  rq_activate_all_grippers(False)
  # end: URCap Program Node
  end
  thread Gripper_Activate_thread():
  Gripper_Activate_definition()
  daemon.done_executing()
  end
  def Gripper_Activate():
  textmsg("Executing event: Gripper_Activate")
  __er_thread_handle = run Gripper_Activate_thread()
  end
  if (not daemon.register_method("Gripper_Activate","[]", False)):
    textmsg("Failed to connect to register method Gripper_Activate")
    halt
  end
  sync()
  # end: URCap Program Node
  # begin: URCap Program Node
  #   Source: EnabledRobotics - ER-ABILITY, 5.0.0, Enabled Robotics ApS
  #   Type: EventNode
  $ 10 "EventNode: Gripper_Open1" "noBreak"
  def Gripper_Open1_definition():
  # begin: URCap Program Node
  #   Source: Robotiq_Grippers, 1.8.13.22852, Robotiq Inc.
  #   Type: Gripper
  $ 11 "Gripper Open (1)" "noBreak"
  if not(gripper_connected[0]):
    popup("Gripper 1 must be connected to run this program.", "No connection", False, True, True)
  end
  if not(rq_is_gripper_activated("1")):
    popup("Gripper 1 is not activated. Go to Installation tab > Gripper to activate it and run the program again.", "Not activated", False, True, True)
  end
  rq_set_pos_spd_for(0, 255, 0, "1")
  rq_wait_pos_spe_for_request(0, 255, 0, "1")
  rq_go_to("1")
  rq_wait("1")
  # end: URCap Program Node
  end
  thread Gripper_Open1_thread():
  Gripper_Open1_definition()
  daemon.done_executing()
  end
  def Gripper_Open1():
  textmsg("Executing event: Gripper_Open1")
  __er_thread_handle = run Gripper_Open1_thread()
  end
  if (not daemon.register_method("Gripper_Open1","[]", False)):
    textmsg("Failed to connect to register method Gripper_Open1")
    halt
  end
  sync()
  # end: URCap Program Node
  # begin: URCap Program Node
  #   Source: EnabledRobotics - ER-ABILITY, 5.0.0, Enabled Robotics ApS
  #   Type: EventNode
  $ 12 "EventNode: Gripper_Close" "noBreak"
  def Gripper_Close_definition():
  # begin: URCap Program Node
  #   Source: Robotiq_Grippers, 1.8.13.22852, Robotiq Inc.
  #   Type: Gripper
  $ 13 "Gripper Close (1)" "noBreak"
  if not(gripper_connected[0]):
    popup("Gripper 1 must be connected to run this program.", "No connection", False, True, True)
  end
  if not(rq_is_gripper_activated("1")):
    popup("Gripper 1 is not activated. Go to Installation tab > Gripper to activate it and run the program again.", "Not activated", False, True, True)
  end
  rq_set_pos_spd_for(255, 255, 0, "1")
  rq_wait_pos_spe_for_request(255, 255, 0, "1")
  rq_go_to("1")
  rq_wait("1")
  # end: URCap Program Node
  end
  thread Gripper_Close_thread():
  Gripper_Close_definition()
  daemon.done_executing()
  end
  def Gripper_Close():
  textmsg("Executing event: Gripper_Close")
  __er_thread_handle = run Gripper_Close_thread()
  end
  if (not daemon.register_method("Gripper_Close","[]", False)):
    textmsg("Failed to connect to register method Gripper_Close")
    halt
  end
  sync()
  # end: URCap Program Node
  # begin: URCap Program Node
  #   Source: EnabledRobotics - ER-ABILITY, 5.0.0, Enabled Robotics ApS
  #   Type: EventNode
  $ 14 "EventNode: Unload" "noBreak"
  global __er_Unload_arg_pose = p[0, 0, 0, 0, 0, 0]
  def Unload_definition(arg_pose):
  $ 15 "Unload_ref≔__er_Unload_arg_pose" "noBreak"
  global Unload_ref=__er_Unload_arg_pose
  $ 16 "MoveJ" "noBreak"
  $ 17 "Waypoint_2" "noBreak"
  movej(get_inverse_kin(Waypoint_2_p, qnear=Waypoint_2_q), a=1.3962634015954636, v=1.0471975511965976)
  $ 18 "Pallet_2" "noBreak"
  def Pallet_2_trans(pose):
  return p[pose[0], pose[1], pose[2], 0, 0, 0]
  end
  def Pallet_2_rot(pose):
  return p[0, 0, 0, pose[3], pose[4], pose[5]]
  end
  def Pallet_2_compute_pallet_waypoint(T_base_feature_taught, T_feature_referencePoint_taught, T_referencePoint_approach_taught, T_base_feature, T_base_referencePoint):
  local trans_referencePoint_approach_in_feature_taught = pose_sub(Pallet_2_trans(pose_trans(T_feature_referencePoint_taught, T_referencePoint_approach_taught)), Pallet_2_trans(T_feature_referencePoint_taught))
  local rot_referencePoint_approach_in_feature_taught = pose_trans(Pallet_2_rot(T_feature_referencePoint_taught), pose_trans(Pallet_2_rot(T_referencePoint_approach_taught), pose_inv(Pallet_2_rot(T_feature_referencePoint_taught))))
  T_feature_referencePoint = pose_trans(pose_inv(T_base_feature), T_base_referencePoint)
  rot_referencePoint_approach = pose_trans(pose_inv(Pallet_2_rot(T_feature_referencePoint)), pose_trans(rot_referencePoint_approach_in_feature_taught, Pallet_2_rot(T_feature_referencePoint)))
  T_feature_approach = pose_trans(trans_referencePoint_approach_in_feature_taught, pose_trans(T_feature_referencePoint, rot_referencePoint_approach))
  T_base_approach = pose_trans(T_base_feature, T_feature_approach)
  return T_base_approach
  end
  Pallet_2_tct_1 = 3
  if (Pallet_2_cnt_1 > 3 or Pallet_2_cnt_1 < 1):
    Pallet_2_cnt_1 = 1
  end
  $ 19 "Patterns" "noBreak"
  $ 20 "Line_Pattern_2" "noBreak"
  $ 23 "Layers" "noBreak"
  if (Pallet_2_cnt_1 < 4):
    Pallet_2_lno_1 = 1
    Pallet_2_lct_1 = Pallet_2_cnt_1
    global StartItem_2=pose_trans(p[0.0,0.0,0.0,0.0,0.0,0.0], pose_trans(p[-.000000000000, -.000000000000, -.000000000000, .000000000000, .000000000000, .000000000000], p[.520226808930, .071936160165, -.439816599331, 3.141509651494, .015551157232, .000010800258]))
    global EndItem_2=pose_trans(p[0.0,0.0,0.0,0.0,0.0,0.0], pose_trans(p[-.000000000000, -.000000000000, -.000000000000, .000000000000, .000000000000, .000000000000], p[.521976506042, -.107892547401, -.439624527362, 3.141328655500, .039596804554, -.000022510547]))
    referencePoint = interpolate_pose(StartItem_2, EndItem_2, (Pallet_2_lct_1 - 1)/2)
    if ((Pallet_2_lct_1 - 1) < 1.5):
      qNearApproach = [2.5448785455331526, 0.32353681292985914, 0.8867449467631632, -1.209835749483231, -0.6015755965885301, -3.1422033514088064]
    else:
      qNearApproach = [2.318553773487707, 0.5230815444746025, 0.3070377710571135, -0.8290774467610227, -0.8454805618969878, -3.143220671816902]
    end
    direction = p[0,0,1,0,0,0]
    referencePoint = pose_add (referencePoint,p[0.0*direction[0],0.0*direction[1],0.0*direction[2],0,0,0])
  end
  Approach_3_p = Pallet_2_compute_pallet_waypoint(p[0.0,0.0,0.0,0.0,0.0,0.0], pose_trans(pose_inv(p[0.0,0.0,0.0,0.0,0.0,0.0]), p[0.52022680893046,0.07193616016490022,-0.4398165993312858,3.1415096514942586,0.01555115723185833,1.080025776929912E-5]), p[-1.5009913569219435E-4,-1.4773289497117814E-4,-0.07363840846726544,4.5745872302844587E-4,-5.141193914981974E-4,-2.8251868715170223E-4], p[0.0,0.0,0.0,0.0,0.0,0.0], referencePoint)
  Approach_3_p = pose_trans(p[0.52022680893046,0.07193616016490022,-0.4398165993312858,3.141509651511718,0.015551157231944729,1.0800257734370728E-5], pose_trans(pose_inv(referencePoint), Approach_3_p))
  Approach_3_q = qNearApproach
  ToolActionPoi_3_p = Pallet_2_compute_pallet_waypoint(p[0.0,0.0,0.0,0.0,0.0,0.0], pose_trans(pose_inv(p[0.0,0.0,0.0,0.0,0.0,0.0]), p[0.52022680893046,0.07193616016490022,-0.4398165993312858,3.1415096514942586,0.01555115723185833,1.080025776929912E-5]), p[-1.1102230246251565E-16,1.3877787807814457E-17,0.0,0.0,0.0,0.0], p[0.0,0.0,0.0,0.0,0.0,0.0], referencePoint)
  ToolActionPoi_3_p = pose_trans(p[0.52022680893046,0.07193616016490022,-0.4398165993312858,3.141509651511718,0.015551157231944729,1.0800257734370728E-5], pose_trans(pose_inv(referencePoint), ToolActionPoi_3_p))
  Exit_4_p = Pallet_2_compute_pallet_waypoint(p[0.0,0.0,0.0,0.0,0.0,0.0], pose_trans(pose_inv(p[0.0,0.0,0.0,0.0,0.0,0.0]), p[0.52022680893046,0.07193616016490022,-0.4398165993312858,3.1415096514942586,0.01555115723185833,1.080025776929912E-5]), p[-3.93932843645306E-6,-7.071115271761741E-6,-0.10081098319262166,2.4279295122529868E-5,-8.605183831750915E-6,-1.5904010148868937E-5], p[0.0,0.0,0.0,0.0,0.0,0.0], referencePoint)
  Exit_4_p = pose_trans(p[0.52022680893046,0.07193616016490022,-0.4398165993312858,3.141509651511718,0.015551157231944729,1.0800257734370728E-5], pose_trans(pose_inv(referencePoint), Exit_4_p))
  $ 24 "At Each Item" "noBreak"
  $ 25 "Generated Movements" "noBreak"
  $ 26 "MoveJ" "noBreak"
  $ 27 "Approach_3" "noBreak"
  movej(get_inverse_kin(pose_trans(referencePoint, pose_trans(p[-.520910568349, .066801880452, -.439817090922, -3.141509651507, -.015551157232, -.000010800258], Approach_3_p)), qnear=Approach_3_q), a=1.3962634015954636, v=1.0471975511965976)
  $ 28 "MoveL" "noBreak"
  $ 29 "ToolActionPoi_3" "noBreak"
  movel(pose_trans(referencePoint, pose_trans(p[-.520910568349, .066801880452, -.439817090922, -3.141509651507, -.015551157232, -.000010800258], ToolActionPoi_3_p)), a=1.2, v=0.25)
  $ 30 "Tool action" "noBreak"
  # begin: URCap Program Node
  #   Source: Robotiq_Grippers, 1.8.13.22852, Robotiq Inc.
  #   Type: Gripper
  $ 31 "Gripper Close (1)" "noBreak"
  if not(gripper_connected[0]):
    popup("Gripper 1 must be connected to run this program.", "No connection", False, True, True)
  end
  if not(rq_is_gripper_activated("1")):
    popup("Gripper 1 is not activated. Go to Installation tab > Gripper to activate it and run the program again.", "Not activated", False, True, True)
  end
  rq_set_pos_spd_for(255, 255, 255, "1")
  rq_wait_pos_spe_for_request(255, 255, 255, "1")
  rq_go_to("1")
  rq_wait("1")
  # end: URCap Program Node
  $ 32 "MoveL" "noBreak"
  $ 33 "Exit_4" "noBreak"
  movel(pose_trans(referencePoint, pose_trans(p[-.520910568349, .066801880452, -.439817090922, -3.141509651507, -.015551157232, -.000010800258], Exit_4_p)), a=1.2, v=0.25)
  Pallet_2_sep_1 = False
  if (Pallet_2_cnt_1 >= 3):
    Pallet_2_cnt_1 = 1
  else:
    Pallet_2_cnt_1 = Pallet_2_cnt_1 + 1
  end
  $ 34 "MoveJ" "noBreak"
  $ 35 "Waypoint_2" "noBreak"
  movej(get_inverse_kin(Waypoint_2_p, qnear=Waypoint_2_q), a=1.3962634015954636, v=1.0471975511965976)
  $ 36 "Pallet_1" "noBreak"
  def Pallet_1_trans(pose):
  return p[pose[0], pose[1], pose[2], 0, 0, 0]
  end
  def Pallet_1_rot(pose):
  return p[0, 0, 0, pose[3], pose[4], pose[5]]
  end
  def Pallet_1_compute_pallet_waypoint(T_base_feature_taught, T_feature_referencePoint_taught, T_referencePoint_approach_taught, T_base_feature, T_base_referencePoint):
  local trans_referencePoint_approach_in_feature_taught = pose_sub(Pallet_1_trans(pose_trans(T_feature_referencePoint_taught, T_referencePoint_approach_taught)), Pallet_1_trans(T_feature_referencePoint_taught))
  local rot_referencePoint_approach_in_feature_taught = pose_trans(Pallet_1_rot(T_feature_referencePoint_taught), pose_trans(Pallet_1_rot(T_referencePoint_approach_taught), pose_inv(Pallet_1_rot(T_feature_referencePoint_taught))))
  T_feature_referencePoint = pose_trans(pose_inv(T_base_feature), T_base_referencePoint)
  rot_referencePoint_approach = pose_trans(pose_inv(Pallet_1_rot(T_feature_referencePoint)), pose_trans(rot_referencePoint_approach_in_feature_taught, Pallet_1_rot(T_feature_referencePoint)))
  T_feature_approach = pose_trans(trans_referencePoint_approach_in_feature_taught, pose_trans(T_feature_referencePoint, rot_referencePoint_approach))
  T_base_approach = pose_trans(T_base_feature, T_feature_approach)
  return T_base_approach
  end
  Pallet_2_tct_2 = 3
  if (Pallet_2_cnt_2 > 3 or Pallet_2_cnt_2 < 1):
    Pallet_2_cnt_2 = 1
  end
  $ 37 "Patterns" "noBreak"
  $ 38 "Line_Pattern_1" "noBreak"
  $ 41 "Layers" "noBreak"
  if (Pallet_2_cnt_2 < 4):
    Pallet_2_lno_2 = 1
    Pallet_2_lct_2 = Pallet_2_cnt_2
    global StartItem_1=pose_trans(Unload_ref, pose_trans(p[-.592420775083, .276699022305, .196891037220, 2.141026582984, -2.289780745210, -.016012414057], p[.145742456500, -.623712299717, .141843363677, -2.162912830523, 2.278464349970, .000016883489]))
    global EndItem_1=pose_trans(Unload_ref, pose_trans(p[-.592420775083, .276699022305, .196891037220, 2.141026582984, -2.289780745210, -.016012414057], p[-.034366509976, -.616405446345, .140307709095, 2.162884038701, -2.278479638159, .000010711089]))
    referencePoin_1 = interpolate_pose(StartItem_1, EndItem_1, (Pallet_2_lct_2 - 1)/2)
    if ((Pallet_2_lct_2 - 1) < 1.5):
      qNearApproach_1 = [1.4717269593278084, -0.377092883754063, 1.1086358557351508, -4.010618644468483, 0.2053468506389249, 0.11347314803018159]
    else:
      qNearApproach_1 = [1.223852267476565, -0.3417190093073499, 1.0145159265446688, -3.879360012423625, 0.4524234852589557, 0.035990198425167035]
    end
    direction = pose_trans(p[0,0,0,Unload_ref[3],Unload_ref[4],Unload_ref[5]], p[0,0,1,0,0,0])
    referencePoin_1 = pose_add (referencePoin_1,p[0.0*direction[0],0.0*direction[1],0.0*direction[2],0,0,0])
  end
  Approach_p = Pallet_1_compute_pallet_waypoint(p[0.23673981765789284,-0.611972183808765,0.18903732227235456,-2.141026582984071,2.2897807452097325,0.016012414057338102], pose_trans(pose_inv(p[0.23673981765789284,-0.611972183808765,0.18903732227235456,-2.141026582984071,2.2897807452097325,0.016012414057338102]), p[0.14574245649996154,-0.6237122997166273,0.14184336367685696,-2.1629128305231067,2.278464349969941,1.688348907601959E-5]), p[0.0011206971510525632,0.0015926661309434986,-0.05760783126324068,0.031976489334781005,-0.019679141912164282,-0.020960074111678773], Unload_ref, referencePoin_1)
  Approach_p = pose_trans(p[0.3302161821107999,-0.6547625956979264,0.14667608988337466,2.3106327262625443,-2.073456813515827,-0.009785998864891442], pose_trans(pose_inv(referencePoin_1), Approach_p))
  Approach_q = qNearApproach_1
  ToolActionPoint_p = Pallet_1_compute_pallet_waypoint(p[0.23673981765789284,-0.611972183808765,0.18903732227235456,-2.141026582984071,2.2897807452097325,0.016012414057338102], pose_trans(pose_inv(p[0.23673981765789284,-0.611972183808765,0.18903732227235456,-2.141026582984071,2.2897807452097325,0.016012414057338102]), p[0.14574245649996154,-0.6237122997166273,0.14184336367685696,-2.1629128305231067,2.278464349969941,1.688348907601959E-5]), p[-0.05091451474589437,0.1798191171068455,0.009530418404298385,0.030088811758342437,-0.022546045786153587,0.16009642489347953], Unload_ref, referencePoin_1)
  ToolActionPoint_p = pose_trans(p[0.3302161821107999,-0.6547625956979264,0.14667608988337466,2.3106327262625443,-2.073456813515827,-0.009785998864891442], pose_trans(pose_inv(referencePoin_1), ToolActionPoint_p))
  Exit_1_p = Pallet_1_compute_pallet_waypoint(p[0.23673981765789284,-0.611972183808765,0.18903732227235456,-2.141026582984071,2.2897807452097325,0.016012414057338102], pose_trans(pose_inv(p[0.23673981765789284,-0.611972183808765,0.18903732227235456,-2.141026582984071,2.2897807452097325,0.016012414057338102]), p[0.14574245649996154,-0.6237122997166273,0.14184336367685696,-2.1629128305231067,2.278464349969941,1.688348907601959E-5]), p[0.0012088044817964994,6.156659549959032E-4,-0.05405850596043982,1.6947789472419606E-5,2.6304475016522655E-5,-6.152303689366298E-6], Unload_ref, referencePoin_1)
  Exit_1_p = pose_trans(p[0.3302161821107999,-0.6547625956979264,0.14667608988337466,2.3106327262625443,-2.073456813515827,-0.009785998864891442], pose_trans(pose_inv(referencePoin_1), Exit_1_p))
  $ 42 "At Each Item" "noBreak"
  $ 43 "Generated Movements" "noBreak"
  $ 44 "MoveJ" "noBreak"
  $ 45 "Approach" "noBreak"
  movej(get_inverse_kin(pose_trans(referencePoin_1, pose_trans(p[-.689448135507, .253081536651, .141002351928, -2.310632726263, 2.073456813516, .009785998865], Approach_p)), qnear=Approach_q), a=1.3962634015954636, v=1.0471975511965976)
  $ 46 "MoveL" "noBreak"
  $ 47 "ToolActionPoint" "noBreak"
  movel(pose_trans(referencePoin_1, pose_trans(p[-.689448135507, .253081536651, .141002351928, -2.310632726263, 2.073456813516, .009785998865], ToolActionPoint_p)), a=1.2, v=0.25)
  $ 48 "Tool action" "noBreak"
  # begin: URCap Program Node
  #   Source: Robotiq_Grippers, 1.8.13.22852, Robotiq Inc.
  #   Type: Gripper
  $ 49 "Gripper Open (1)" "noBreak"
  if not(gripper_connected[0]):
    popup("Gripper 1 must be connected to run this program.", "No connection", False, True, True)
  end
  if not(rq_is_gripper_activated("1")):
    popup("Gripper 1 is not activated. Go to Installation tab > Gripper to activate it and run the program again.", "Not activated", False, True, True)
  end
  rq_set_pos_spd_for(0, 255, 255, "1")
  rq_wait_pos_spe_for_request(0, 255, 255, "1")
  rq_go_to("1")
  rq_wait("1")
  # end: URCap Program Node
  $ 50 "MoveL" "noBreak"
  $ 51 "Exit_1" "noBreak"
  movel(pose_trans(referencePoin_1, pose_trans(p[-.689448135507, .253081536651, .141002351928, -2.310632726263, 2.073456813516, .009785998865], Exit_1_p)), a=1.2, v=0.25)
  Pallet_2_sep_2 = False
  if (Pallet_2_cnt_2 >= 3):
    Pallet_2_cnt_2 = 1
  else:
    Pallet_2_cnt_2 = Pallet_2_cnt_2 + 1
  end
  $ 52 "MoveJ" "noBreak"
  $ 53 "Waypoint_2" "noBreak"
  movej(get_inverse_kin(Waypoint_2_p, qnear=Waypoint_2_q), a=1.3962634015954636, v=1.0471975511965976)
  end
  thread Unload_thread():
  Unload_definition(__er_Unload_arg_pose)
  daemon.done_executing()
  end
  def Unload(arg_pose):
  textmsg("Executing event: Unload, with arguments:")
  textmsg("Argument: arg_pose = ", arg_pose)
  __er_Unload_arg_pose = arg_pose
  __er_thread_handle = run Unload_thread()
  end
  if (not daemon.register_method("Unload","[pose]", False)):
    textmsg("Failed to connect to register method Unload")
    halt
  end
  sync()
  # end: URCap Program Node
  # begin: URCap Program Node
  #   Source: EnabledRobotics - ER-ABILITY, 5.0.0, Enabled Robotics ApS
  #   Type: EventNode
  $ 54 "EventNode: Palletize" "noBreak"
  global __er_Palletize_arg_pose = p[0, 0, 0, 0, 0, 0]
  def Palletize_definition(arg_pose):
  $ 55 "Pallet_ref≔__er_Palletize_arg_pose" "noBreak"
  global Pallet_ref=__er_Palletize_arg_pose
  $ 56 "MoveJ" "noBreak"
  $ 58 "Waypoint_2" "noBreak"
  movej(get_inverse_kin(Waypoint_2_p, qnear=Waypoint_2_q), a=1.3962634015954636, v=1.0471975511965976)
  $ 59 "Pallet_3" "noBreak"
  def Pallet_3_trans(pose):
  return p[pose[0], pose[1], pose[2], 0, 0, 0]
  end
  def Pallet_3_rot(pose):
  return p[0, 0, 0, pose[3], pose[4], pose[5]]
  end
  def Pallet_3_compute_pallet_waypoint(T_base_feature_taught, T_feature_referencePoint_taught, T_referencePoint_approach_taught, T_base_feature, T_base_referencePoint):
  local trans_referencePoint_approach_in_feature_taught = pose_sub(Pallet_3_trans(pose_trans(T_feature_referencePoint_taught, T_referencePoint_approach_taught)), Pallet_3_trans(T_feature_referencePoint_taught))
  local rot_referencePoint_approach_in_feature_taught = pose_trans(Pallet_3_rot(T_feature_referencePoint_taught), pose_trans(Pallet_3_rot(T_referencePoint_approach_taught), pose_inv(Pallet_3_rot(T_feature_referencePoint_taught))))
  T_feature_referencePoint = pose_trans(pose_inv(T_base_feature), T_base_referencePoint)
  rot_referencePoint_approach = pose_trans(pose_inv(Pallet_3_rot(T_feature_referencePoint)), pose_trans(rot_referencePoint_approach_in_feature_taught, Pallet_3_rot(T_feature_referencePoint)))
  T_feature_approach = pose_trans(trans_referencePoint_approach_in_feature_taught, pose_trans(T_feature_referencePoint, rot_referencePoint_approach))
  T_base_approach = pose_trans(T_base_feature, T_feature_approach)
  return T_base_approach
  end
  Pallet_2_tct_3 = 3
  if (Pallet_2_cnt_3 > 3 or Pallet_2_cnt_3 < 1):
    Pallet_2_cnt_3 = 1
  end
  $ 60 "Patterns" "noBreak"
  $ 61 "Line_Pattern_5" "noBreak"
  $ 64 "Layers" "noBreak"
  if (Pallet_2_cnt_3 < 4):
    Pallet_2_lno_3 = 1
    Pallet_2_lct_3 = Pallet_2_cnt_3
    global StartItem_5=pose_trans(Pallet_ref, pose_trans(p[-.592420775083, .276699022305, .196891037220, 2.141026582984, -2.289780745210, -.016012414057], p[.145742456500, -.623712299717, .141843363677, -2.162912830523, 2.278464349970, .000016883489]))
    global EndItem_5=pose_trans(Pallet_ref, pose_trans(p[-.592420775083, .276699022305, .196891037220, 2.141026582984, -2.289780745210, -.016012414057], p[-.034364587449, -.616414812009, .134803893258, 2.162884771053, -2.278474941594, .000025529303]))
    referencePoin_6 = interpolate_pose(StartItem_5, EndItem_5, (Pallet_2_lct_3 - 1)/2)
    if ((Pallet_2_lct_3 - 1) < 1.5):
      qNearApproach_2 = [1.160836153948624, -0.48475985649287523, 1.429198472833832, -4.07612878433148, 0.3533404294143797, -0.011125824810111595]
    else:
      qNearApproach_2 = [0.9092989459402957, -0.3906363918532989, 1.217352351317741, -3.9632834025255583, 0.6055194004184299, -0.00720924811746837]
    end
    direction = pose_trans(p[0,0,0,Pallet_ref[3],Pallet_ref[4],Pallet_ref[5]], p[0,0,1,0,0,0])
    referencePoin_6 = pose_add (referencePoin_6,p[0.0*direction[0],0.0*direction[1],0.0*direction[2],0,0,0])
  end
  Approach_2_p = Pallet_3_compute_pallet_waypoint(p[0.23673981765789284,-0.611972183808765,0.18903732227235456,-2.141026582984071,2.2897807452097325,0.016012414057338102], pose_trans(pose_inv(p[0.23673981765789284,-0.611972183808765,0.18903732227235456,-2.141026582984071,2.2897807452097325,0.016012414057338102]), p[0.14574245649996154,-0.6237122997166273,0.14184336367685696,-2.1629128305231067,2.278464349969941,1.688348907601959E-5]), p[-8.821036119655012E-6,9.83391916484222E-6,-0.05174217287322935,-7.92077343834213E-7,-8.53904463359664E-6,4.718218270382111E-6], Pallet_ref, referencePoin_6)
  Approach_2_p = pose_trans(p[0.14574245649996245,-0.6237122997166271,0.14184336367685513,-2.162912830525248,2.2784643499679076,1.6883689364664383E-5], pose_trans(pose_inv(referencePoin_6), Approach_2_p))
  Approach_2_q = qNearApproach_2
  ToolActionPoi_2_p = Pallet_3_compute_pallet_waypoint(p[0.23673981765789284,-0.611972183808765,0.18903732227235456,-2.141026582984071,2.2897807452097325,0.016012414057338102], pose_trans(pose_inv(p[0.23673981765789284,-0.611972183808765,0.18903732227235456,-2.141026582984071,2.2897807452097325,0.016012414057338102]), p[0.14574245649996154,-0.6237122997166273,0.14184336367685696,-2.1629128305231067,2.278464349969941,1.688348907601959E-5]), p[2.220446049250313E-16,9.159339953157541E-16,-1.8318679906315083E-15,0.0,0.0,0.0], Pallet_ref, referencePoin_6)
  ToolActionPoi_2_p = pose_trans(p[0.14574245649996245,-0.6237122997166271,0.14184336367685513,-2.162912830525248,2.2784643499679076,1.6883689364664383E-5], pose_trans(pose_inv(referencePoin_6), ToolActionPoi_2_p))
  Exit_3_p = Pallet_3_compute_pallet_waypoint(p[0.23673981765789284,-0.611972183808765,0.18903732227235456,-2.141026582984071,2.2897807452097325,0.016012414057338102], pose_trans(pose_inv(p[0.23673981765789284,-0.611972183808765,0.18903732227235456,-2.141026582984071,2.2897807452097325,0.016012414057338102]), p[0.14574245649996154,-0.6237122997166273,0.14184336367685696,-2.1629128305231067,2.278464349969941,1.688348907601959E-5]), p[-4.6349033265835615E-6,6.324703609672522E-6,-0.06181962181018885,-2.875197051692597E-6,-4.847655252132371E-5,1.897897991802547E-5], Pallet_ref, referencePoin_6)
  Exit_3_p = pose_trans(p[0.33020295134031996,-0.6550358453350454,0.14679715883248884,2.3097137152461533,-2.071977896073306,-0.009558990049756003], pose_trans(pose_inv(referencePoin_6), Exit_3_p))
  $ 65 "At Each Item" "noBreak"
  $ 66 "Generated Movements" "noBreak"
  $ 67 "MoveJ" "noBreak"
  $ 68 "Approach_2" "noBreak"
  movej(get_inverse_kin(pose_trans(referencePoin_6, pose_trans(p[-.615288801215, .177976730796, .141849958260, 2.162912830677, -2.278464350127, -.000016883689], Approach_2_p)), qnear=Approach_2_q), a=1.3962634015954636, v=1.0471975511965976)
  $ 69 "MoveL" "noBreak"
  $ 70 "ToolActionPoi_2" "noBreak"
  movel(pose_trans(referencePoin_6, pose_trans(p[-.615288801215, .177976730796, .141849958260, 2.162912830677, -2.278464350127, -.000016883689], ToolActionPoi_2_p)), a=1.2, v=0.25)
  $ 71 "Tool action" "noBreak"
  # begin: URCap Program Node
  #   Source: Robotiq_Grippers, 1.8.13.22852, Robotiq Inc.
  #   Type: Gripper
  $ 72 "Gripper Close (1)" "noBreak"
  if not(gripper_connected[0]):
    popup("Gripper 1 must be connected to run this program.", "No connection", False, True, True)
  end
  if not(rq_is_gripper_activated("1")):
    popup("Gripper 1 is not activated. Go to Installation tab > Gripper to activate it and run the program again.", "Not activated", False, True, True)
  end
  rq_set_pos_spd_for(255, 153, 56, "1")
  rq_wait_pos_spe_for_request(255, 153, 56, "1")
  rq_go_to("1")
  rq_wait("1")
  # end: URCap Program Node
  $ 73 "MoveL" "noBreak"
  $ 74 "Exit_3" "noBreak"
  movel(pose_trans(referencePoin_6, pose_trans(p[-.689971033309, .252662774639, .140559059103, -2.309713715246, 2.071977896073, .009558990050], Exit_3_p)), a=1.2, v=0.25)
  Pallet_2_sep_3 = False
  if (Pallet_2_cnt_3 >= 3):
    Pallet_2_cnt_3 = 1
  else:
    Pallet_2_cnt_3 = Pallet_2_cnt_3 + 1
  end
  $ 75 "MoveJ" "noBreak"
  $ 76 "Waypoint_2" "noBreak"
  movej(get_inverse_kin(Waypoint_2_p, qnear=Waypoint_2_q), a=1.3962634015954636, v=1.0471975511965976)
  $ 77 "Pallet_4" "noBreak"
  def Pallet_4_trans(pose):
  return p[pose[0], pose[1], pose[2], 0, 0, 0]
  end
  def Pallet_4_rot(pose):
  return p[0, 0, 0, pose[3], pose[4], pose[5]]
  end
  def Pallet_4_compute_pallet_waypoint(T_base_feature_taught, T_feature_referencePoint_taught, T_referencePoint_approach_taught, T_base_feature, T_base_referencePoint):
  local trans_referencePoint_approach_in_feature_taught = pose_sub(Pallet_4_trans(pose_trans(T_feature_referencePoint_taught, T_referencePoint_approach_taught)), Pallet_4_trans(T_feature_referencePoint_taught))
  local rot_referencePoint_approach_in_feature_taught = pose_trans(Pallet_4_rot(T_feature_referencePoint_taught), pose_trans(Pallet_4_rot(T_referencePoint_approach_taught), pose_inv(Pallet_4_rot(T_feature_referencePoint_taught))))
  T_feature_referencePoint = pose_trans(pose_inv(T_base_feature), T_base_referencePoint)
  rot_referencePoint_approach = pose_trans(pose_inv(Pallet_4_rot(T_feature_referencePoint)), pose_trans(rot_referencePoint_approach_in_feature_taught, Pallet_4_rot(T_feature_referencePoint)))
  T_feature_approach = pose_trans(trans_referencePoint_approach_in_feature_taught, pose_trans(T_feature_referencePoint, rot_referencePoint_approach))
  T_base_approach = pose_trans(T_base_feature, T_feature_approach)
  return T_base_approach
  end
  Pallet_2_tct_4 = 3
  if (Pallet_2_cnt_4 > 3 or Pallet_2_cnt_4 < 1):
    Pallet_2_cnt_4 = 1
  end
  $ 78 "Patterns" "noBreak"
  $ 79 "Line_Pattern_6" "noBreak"
  $ 82 "Layers" "noBreak"
  if (Pallet_2_cnt_4 < 4):
    Pallet_2_lno_4 = 1
    Pallet_2_lct_4 = Pallet_2_cnt_4
    global StartItem_6=pose_trans(p[0.0,0.0,0.0,0.0,0.0,0.0], pose_trans(p[-.000000000000, -.000000000000, -.000000000000, .000000000000, .000000000000, .000000000000], p[.520226808930, .071936160165, -.439816599331, 3.141509651494, .015551157232, .000010800258]))
    global EndItem_6=pose_trans(p[0.0,0.0,0.0,0.0,0.0,0.0], pose_trans(p[-.000000000000, -.000000000000, -.000000000000, .000000000000, .000000000000, .000000000000], p[.521976506042, -.107892547401, -.439624527362, 3.141328655500, .039596804554, -.000022510547]))
    referencePoin_7 = interpolate_pose(StartItem_6, EndItem_6, (Pallet_2_lct_4 - 1)/2)
    if ((Pallet_2_lct_4 - 1) < 1.5):
      qNearApproach_3 = [2.5448785455331526, 0.32353681292985914, 0.8867449467631632, -1.209835749483231, -0.6015755965885301, -3.1422033514088064]
    else:
      qNearApproach_3 = [2.318553773487707, 0.5230815444746025, 0.3070377710571135, -0.8290774467610227, -0.8454805618969878, -3.143220671816902]
    end
    direction = p[0,0,1,0,0,0]
    referencePoin_7 = pose_add (referencePoin_7,p[0.0*direction[0],0.0*direction[1],0.0*direction[2],0,0,0])
  end
  Approach_3_p = Pallet_4_compute_pallet_waypoint(p[0.0,0.0,0.0,0.0,0.0,0.0], pose_trans(pose_inv(p[0.0,0.0,0.0,0.0,0.0,0.0]), p[0.52022680893046,0.07193616016490022,-0.4398165993312858,3.1415096514942586,0.01555115723185833,1.080025776929912E-5]), p[-1.5009913569219435E-4,-1.4773289497117814E-4,-0.07363840846726544,4.5745872302844587E-4,-5.141193914981974E-4,-2.8251868715170223E-4], p[0.0,0.0,0.0,0.0,0.0,0.0], referencePoin_7)
  Approach_3_p = pose_trans(p[0.52022680893046,0.07193616016490022,-0.4398165993312858,3.141509651511718,0.015551157231944729,1.0800257734370728E-5], pose_trans(pose_inv(referencePoin_7), Approach_3_p))
  Approach_3_q = qNearApproach_3
  ToolActionPoi_3_p = Pallet_4_compute_pallet_waypoint(p[0.0,0.0,0.0,0.0,0.0,0.0], pose_trans(pose_inv(p[0.0,0.0,0.0,0.0,0.0,0.0]), p[0.52022680893046,0.07193616016490022,-0.4398165993312858,3.1415096514942586,0.01555115723185833,1.080025776929912E-5]), p[-1.1102230246251565E-16,1.3877787807814457E-17,0.0,0.0,0.0,0.0], p[0.0,0.0,0.0,0.0,0.0,0.0], referencePoin_7)
  ToolActionPoi_3_p = pose_trans(p[0.52022680893046,0.07193616016490022,-0.4398165993312858,3.141509651511718,0.015551157231944729,1.0800257734370728E-5], pose_trans(pose_inv(referencePoin_7), ToolActionPoi_3_p))
  Exit_4_p = Pallet_4_compute_pallet_waypoint(p[0.0,0.0,0.0,0.0,0.0,0.0], pose_trans(pose_inv(p[0.0,0.0,0.0,0.0,0.0,0.0]), p[0.52022680893046,0.07193616016490022,-0.4398165993312858,3.1415096514942586,0.01555115723185833,1.080025776929912E-5]), p[-3.93932843645306E-6,-7.071115271761741E-6,-0.10081098319262166,2.4279295122529868E-5,-8.605183831750915E-6,-1.5904010148868937E-5], p[0.0,0.0,0.0,0.0,0.0,0.0], referencePoin_7)
  Exit_4_p = pose_trans(p[0.52022680893046,0.07193616016490022,-0.4398165993312858,3.141509651511718,0.015551157231944729,1.0800257734370728E-5], pose_trans(pose_inv(referencePoin_7), Exit_4_p))
  $ 83 "At Each Item" "noBreak"
  $ 84 "Generated Movements" "noBreak"
  $ 85 "MoveJ" "noBreak"
  $ 86 "Approach_3" "noBreak"
  movej(get_inverse_kin(pose_trans(referencePoin_7, pose_trans(p[-.520910568349, .066801880452, -.439817090922, -3.141509651507, -.015551157232, -.000010800258], Approach_3_p)), qnear=Approach_3_q), a=1.3962634015954636, v=1.0471975511965976)
  $ 87 "MoveL" "noBreak"
  $ 88 "ToolActionPoi_3" "noBreak"
  movel(pose_trans(referencePoin_7, pose_trans(p[-.520910568349, .066801880452, -.439817090922, -3.141509651507, -.015551157232, -.000010800258], ToolActionPoi_3_p)), a=1.2, v=0.25)
  $ 89 "Tool action" "noBreak"
  # begin: URCap Program Node
  #   Source: Robotiq_Grippers, 1.8.13.22852, Robotiq Inc.
  #   Type: Gripper
  $ 90 "Gripper Open (1)" "noBreak"
  if not(gripper_connected[0]):
    popup("Gripper 1 must be connected to run this program.", "No connection", False, True, True)
  end
  if not(rq_is_gripper_activated("1")):
    popup("Gripper 1 is not activated. Go to Installation tab > Gripper to activate it and run the program again.", "Not activated", False, True, True)
  end
  rq_set_pos_spd_for(0, 153, 56, "1")
  rq_wait_pos_spe_for_request(0, 153, 56, "1")
  rq_go_to("1")
  rq_wait("1")
  # end: URCap Program Node
  $ 91 "MoveL" "noBreak"
  $ 92 "Exit_4" "noBreak"
  movel(pose_trans(referencePoin_7, pose_trans(p[-.520910568349, .066801880452, -.439817090922, -3.141509651507, -.015551157232, -.000010800258], Exit_4_p)), a=1.2, v=0.25)
  Pallet_2_sep_4 = False
  if (Pallet_2_cnt_4 >= 3):
    Pallet_2_cnt_4 = 1
  else:
    Pallet_2_cnt_4 = Pallet_2_cnt_4 + 1
  end
  $ 93 "MoveJ" "noBreak"
  $ 94 "Waypoint_2" "noBreak"
  movej(get_inverse_kin(Waypoint_2_p, qnear=Waypoint_2_q), a=1.3962634015954636, v=1.0471975511965976)
  end
  thread Palletize_thread():
  Palletize_definition(__er_Palletize_arg_pose)
  daemon.done_executing()
  end
  def Palletize(arg_pose):
  textmsg("Executing event: Palletize, with arguments:")
  textmsg("Argument: arg_pose = ", arg_pose)
  __er_Palletize_arg_pose = arg_pose
  __er_thread_handle = run Palletize_thread()
  end
  if (not daemon.register_method("Palletize","[pose]", False)):
    textmsg("Failed to connect to register method Palletize")
    halt
  end
  sync()
  # end: URCap Program Node
  daemon.end_method_registration()
  daemon.set_init_status(2)
  interpreter_mode(clearQueueOnEnter=False)
  # end: URCap Program Node
  end
end
